# EPICS substitutions: depo-orig/depoApp/Db/Oxford_E500.substitutions
file Oxford_E500.template { pattern
{ Sys	, Dev		, Cntl		,PORT		, Chan	}
{ Depo	, "{TC:1}"	, "{TM:1}"	, Depo_TM1	, 1	}
}
